// TwinCAT 3 PLC project Stream_lib
// Title: Stream_lib
// Company: Chua Siang Poh
// Author: Chua Siang Poh
// ProjectVersion: 1.1
// ProgramVersion: 3.1.4020.10
// libraries:
//   Tc2_Standard, * (Beckhoff Automation GmbH)
//   Tc2_System, * (Beckhoff Automation GmbH)
//   Tc3_Module, * (Beckhoff Automation GmbH)
// project tree:
//   Base Component/Class/Binary/ C_BINARYREADER.TcPOU, C_BINARYWRITER.TcPOU
//   Base Component/Class/HTTP/Datatype/ E_HTTP_CODEGROUP.TcDUT, E_HTTP_CONNECTION.TcDUT, E_HTTP_VERB.TcDUT, T_HTTP_BODY.TcDUT, T_HTTP_URL.TcDUT
//   Base Component/Class/HTTP/Functions/ GET_URL_LENGTH.TcPOU
//   Base Component/Class/HTTP/ GVL_HTTP_PARAMETERS.TcGVL
//   Base Component/Class/HTTP/Message/Base/ C_HTTP_MESSAGE.TcPOU
//   Base Component/Class/HTTP/Message/ C_HTTP_HEADER.TcPOU, C_HTTP_REQUEST.TcPOU, C_HTTP_RESPONSE.TcPOU
//   Base Component/Class/Stream/ C_BINARYSTREAM.TcPOU, C_FILESTREAM.TcPOU, C_HTTPSTREAM.TcPOU
//   Base Component/Datatype/ E_STREAMSEEKTYPE.TcDUT
//   Base Component/Interface/ I_STREAM.TcIO
//   Project Information/ F_GetCompany.TcPOU, F_GetTitle.TcPOU, F_GetVersion.TcPOU
//   Version/ Global_Version.TcGVL
// (motion and I/O tree: see PLC project motion_library)
// real-time tasks:
//   TASK PlcTask: cycle T#10ms, priority 20, ADS port 350

// ---- Base Component/Class/HTTP/Datatype/E_HTTP_CODEGROUP.TcDUT
{attribute 'qualified_only'}
{attribute 'strict'}
TYPE E_HTTP_CODEGROUP :
(
	E_GROUP_INFOMATION := 100,
	E_GROUP_SUCCESS := 200,
	E_GROUP_REDIRECTION := 300,
	E_GROUP_CLIENTERROR := 400,
	E_GROUP_SERVERERROR := 500
)UDINT;
END_TYPE

// ---- Base Component/Class/HTTP/Datatype/E_HTTP_CONNECTION.TcDUT
{attribute 'qualified_only'}
{attribute 'strict'}
TYPE E_HTTP_CONNECTION :
(
	E_CONNECTION_CLOSE := 0,
	E_CONNECTION_KEEP_ALIVE
);
END_TYPE

// ---- Base Component/Class/HTTP/Datatype/E_HTTP_VERB.TcDUT
{attribute 'qualified_only'}
{attribute 'strict'}
TYPE E_HTTP_VERB :
(
	E_HTTP_REQUEST_GET := 0,
	E_HTTP_REQUEST_POST,
	E_HTTP_REQUEST_DELETE,
	E_HTTP_REQUEST_PUT,
	E_HTTP_REQUEST_HEAD,
	E_HTTP_REQUEST_CONNECT,
	E_HTTP_REQUEST_OPTIONS,
	E_HTTP_REQUEST_TRACE
)UDINT;
END_TYPE

// ---- Base Component/Class/HTTP/Datatype/T_HTTP_BODY.TcDUT
TYPE T_HTTP_BODY : ARRAY[0..GVL_HTTP_PARAMETERS.MAX_HTTP_BODY_LENGTH] OF BYTE; END_TYPE

// ---- Base Component/Class/HTTP/Datatype/T_HTTP_URL.TcDUT
TYPE T_HTTP_URL : STRING(GVL_HTTP_PARAMETERS.MAX_HTTP_URL_LENGTH); END_TYPE

// ---- Base Component/Datatype/E_STREAMSEEKTYPE.TcDUT
{attribute 'qualified_only'}
{attribute 'strict'}
TYPE E_STREAMSEEKTYPE :
(
	Origin := 0,
	Current,
	End
);
END_TYPE

// ---- Base Component/Class/HTTP/GVL_HTTP_PARAMETERS.TcGVL
{attribute 'qualified_only'}
VAR_GLOBAL CONSTANT
	MAX_HTTP_BODY_LENGTH 	: UDINT := 30000;
	MAX_HTTP_URL_LENGTH 	: UDINT := 1000;
END_VAR

// ---- Version/Global_Version.TcGVL
{attribute 'TcGenerated'}
// This function has been automatically generated from the project information.
VAR_GLOBAL CONSTANT
	{attribute 'const_non_replaced'}
	{attribute 'linkalways'}
	stLibVersion_Stream_lib : ST_LibVersion := (iMajor := 1, iMinor := 1, iBuild := 0, iRevision := 0, sVersion := '1.1');
END_VAR

// ---- Base Component/Interface/I_STREAM.TcIO
INTERFACE I_STREAM

PROPERTY BufferSize : UDINT
GET
END_GET
END_PROPERTY

METHOD Close : DINT
VAR_INPUT
END_VAR
END_METHOD

PROPERTY EndOfStream : BOOL
GET
END_GET
END_PROPERTY

PROPERTY IsValid : BOOL
GET
END_GET
END_PROPERTY

METHOD Peek : DINT
VAR_INPUT
	ptr_DataOut : POINTER TO BYTE;
END_VAR
END_METHOD

PROPERTY Position : UDINT
GET
END_GET
END_PROPERTY

METHOD Read : DINT
VAR_INPUT
	ptr_DataOut : PVOID;
	Length		: UDINT;
END_VAR
END_METHOD

METHOD Seek : DINT
VAR_INPUT
	Offset 		: UDINT;
	SeekStyle 	: E_STREAMSEEKTYPE;
END_VAR
END_METHOD

METHOD Write : DINT
VAR_INPUT
	ptr_DataIn	: PVOID;
	Length		: UDINT;
END_VAR
END_METHOD

END_INTERFACE

// ---- Base Component/Class/Binary/C_BINARYREADER.TcPOU
FUNCTION_BLOCK C_BINARYREADER
VAR_INPUT
END_VAR
VAR_OUTPUT
END_VAR
VAR
	_BASESTREAM 	: I_STREAM;
END_VAR

PROPERTY BASE_STREAM : I_STREAM
GET
Base_Stream := _BASESTREAM;
END_GET
END_PROPERTY

METHOD CLOSE : DINT
VAR_INPUT
END_VAR
Close := _BASESTREAM.Close();
_BASESTREAM := 0;
RETURN;
END_METHOD

METHOD NEW : DINT
VAR_INPUT
	STREAM : I_STREAM;
END_VAR
IF STREAM = 0 THEN
	New := 1;
	RETURN;
ELSE
	IF STREAM.IsValid THEN
		_BASESTREAM := STREAM;
		_BASESTREAM.Seek( 0, E_STREAMSEEKTYPE.Origin);
		New := -1;
		RETURN;
	ELSE
		New := 1;
		RETURN;
	END_IF
END_IF
END_METHOD

METHOD READ_BOOL : DINT
VAR_INPUT
	out_data : POINTER TO BOOL;
END_VAR
IF _BASESTREAM = 0 THEN
	Read_Bool := 1;
	RETURN;
END_IF

Read_Bool := _BASESTREAM.Read(out_data , 1);
RETURN;
END_METHOD

METHOD READ_BYTES : DINT
VAR_INPUT
	out_data 	: POINTER TO BYTE;
	length		: UDINT;
END_VAR
IF _BASESTREAM = 0 THEN
	Read_Bytes := 1;
	RETURN;
END_IF

Read_Bytes := _BASESTREAM.Read(out_data, length);
RETURN;
END_METHOD

METHOD READ_DOUBLE : DINT
VAR_INPUT
	out_data : POINTER TO LREAL;
END_VAR
IF _BASESTREAM = 0 THEN
	Read_Double := 1;
	RETURN;
END_IF

Read_Double := _BASESTREAM.Read(out_data , 8);
RETURN;
END_METHOD

METHOD READ_FLOAT : DINT
VAR_INPUT
	out_data : POINTER TO REAL;
END_VAR
IF _BASESTREAM = 0 THEN
	Read_Float := 1;
	RETURN;
END_IF

Read_Float := _BASESTREAM.Read(out_data , 4);
RETURN;
END_METHOD

METHOD READ_INT16 : DINT
VAR_INPUT
	out_data : POINTER TO INT;
END_VAR
IF _BASESTREAM = 0 THEN
	Read_Int16 := 1;
	RETURN;
END_IF

Read_Int16 := _BASESTREAM.Read(out_data , 2);
RETURN;
END_METHOD

METHOD READ_INT32 : DINT
VAR_INPUT
	out_data : POINTER TO DINT;
END_VAR
IF _BASESTREAM = 0 THEN
	Read_Int32 := 1;
	RETURN;
END_IF

Read_Int32 := _BASESTREAM.Read(out_data , 4);
RETURN;
END_METHOD

METHOD READ_STRING : DINT
VAR_INPUT
	out_data 	: PVOID;
	length		: UDINT;
END_VAR
IF _BASESTREAM = 0 THEN
	Read_String := 1;
	RETURN;
END_IF

Read_String := _BASESTREAM.Read(out_data, length);
RETURN;
END_METHOD

METHOD READ_UINT16 : DINT
VAR_INPUT
	out_data : POINTER TO UINT;
END_VAR
IF _BASESTREAM = 0 THEN
	Read_UInt16 := 1;
	RETURN;
END_IF

Read_UInt16 := _BASESTREAM.Read(out_data , 4);
RETURN;
END_METHOD

METHOD READ_UINT32 : DINT
VAR_INPUT
	out_data : POINTER TO UDINT;
END_VAR
IF _BASESTREAM = 0 THEN
	Read_UInt32 := 1;
	RETURN;
END_IF

Read_UInt32 := _BASESTREAM.Read(out_data , 4);
RETURN;
END_METHOD

END_FUNCTION_BLOCK

// ---- Base Component/Class/Binary/C_BINARYWRITER.TcPOU
FUNCTION_BLOCK C_BINARYWRITER
VAR_INPUT
END_VAR
VAR_OUTPUT
END_VAR
VAR
	_BASESTREAM 	: I_STREAM;
END_VAR

PROPERTY BASE_STREAM : I_STREAM
GET
Base_Stream := _BASESTREAM;
END_GET
END_PROPERTY

METHOD CLOSE : DINT
VAR_INPUT
END_VAR
Close := _BASESTREAM.Close();
_BASESTREAM := 0;
RETURN;
END_METHOD

METHOD NEW : DINT
VAR_INPUT
	STREAM : I_STREAM;
END_VAR
IF STREAM = 0 THEN
	New := 1;
	RETURN;
ELSE
	IF STREAM.IsValid THEN
		_BASESTREAM := STREAM;
		_BASESTREAM.Seek( 0, E_STREAMSEEKTYPE.Origin);
		New := -1;
		RETURN;
	ELSE
		New := 1;
		RETURN;
	END_IF
END_IF
END_METHOD

METHOD WRITE_BOOL : DINT
VAR_INPUT
	in_data : BOOL;
END_VAR
IF _BASESTREAM = 0 THEN
	Write_Bool := 1;
	RETURN;
END_IF

Write_Bool := _BASESTREAM.Write(ADR(in_data), 1);
RETURN;
END_METHOD

METHOD WRITE_BYTES : DINT
VAR_INPUT
	in_data 	: POINTER TO BYTE;
	length		: UDINT;
END_VAR
IF _BASESTREAM = 0 THEN
	Write_Bytes := 1;
	RETURN;
END_IF

Write_Bytes := _BASESTREAM.Write(in_data, length);
RETURN;
END_METHOD

METHOD WRITE_DOUBLE : DINT
VAR_INPUT
	in_data : LREAL;
END_VAR
IF _BASESTREAM = 0 THEN
	Write_Double := 1;
	RETURN;
END_IF

Write_Double := _BASESTREAM.Write(ADR(in_data), 8);
RETURN;
END_METHOD

METHOD WRITE_FLOAT : DINT
VAR_INPUT
	in_data : REAL;
END_VAR
IF _BASESTREAM = 0 THEN
	Write_Float := 1;
	RETURN;
END_IF

Write_Float := _BASESTREAM.Write(ADR(in_data) , 4);
RETURN;
END_METHOD

METHOD WRITE_INT16 : DINT
VAR_INPUT
	in_data : INT;
END_VAR
IF _BASESTREAM = 0 THEN
	Write_Int16 := 1;
	RETURN;
END_IF

Write_Int16 := _BASESTREAM.Write(ADR(in_data) , 2);
RETURN;
END_METHOD

METHOD WRITE_INT32 : DINT
VAR_INPUT
	in_data : DINT;
END_VAR
IF _BASESTREAM = 0 THEN
	Write_Int32 := 1;
	RETURN;
END_IF

Write_Int32 := _BASESTREAM.Write(ADR(in_data) , 4);
RETURN;
END_METHOD

METHOD WRITE_STRING : DINT
VAR_INPUT
	in_data 	: PVOID;
	length		: UDINT;
END_VAR
IF _BASESTREAM = 0 THEN
	Write_String := 1;
	RETURN;
END_IF

Write_String := _BASESTREAM.Write(in_data, length);
RETURN;
END_METHOD

METHOD WRITE_UINT16 : DINT
VAR_INPUT
	in_data : UINT;
END_VAR
IF _BASESTREAM = 0 THEN
	Write_UInt16 := 1;
	RETURN;
END_IF

Write_UInt16 := _BASESTREAM.Write(ADR(in_data) , 4);
RETURN;
END_METHOD

METHOD WRITE_UINT32 : DINT
VAR_INPUT
	in_data : UDINT;
END_VAR
IF _BASESTREAM = 0 THEN
	Write_UInt32 := 1;
	RETURN;
END_IF

Write_UInt32 := _BASESTREAM.Write(ADR(in_data) , 4);
RETURN;
END_METHOD

END_FUNCTION_BLOCK

// ---- Base Component/Class/HTTP/Functions/GET_URL_LENGTH.TcPOU
FUNCTION GET_URL_LENGTH : UDINT
VAR_INPUT
	PTR_URL : POINTER TO BYTE;
END_VAR
VAR
	I : UDINT;
END_VAR

FOR I := 0 TO GVL_HTTP_PARAMETERS.MAX_HTTP_URL_LENGTH BY 1 DO
	IF PTR_URL[I] = 0 THEN
		GET_URL_LENGTH := I;
		RETURN;
	END_IF
END_FOR
GET_URL_LENGTH := 0;
RETURN;

END_FUNCTION

// ---- Base Component/Class/HTTP/Message/Base/C_HTTP_MESSAGE.TcPOU
FUNCTION_BLOCK C_HTTP_MESSAGE
VAR_INPUT
END_VAR
VAR_OUTPUT
END_VAR
VAR
	//General header
		_CONNECTION 		: E_HTTP_CONNECTION;
	(*
		_CACHE_CONTROL		: STRING(255);
		_DATE 				: STRING(255);
		_PRAGMA				: STRING(255);
		_TRAILER 			: STRING(255);
		_TRANSFER_ENCODING	: STRING(255);
		_UPGRADE 			: STRING(255);
		_VIA 				: STRING(255);
		_WARNING 			: STRING(255);
	*)
	//Entity header
		_CONTENT_LENGTH		: UDINT;
	(*
		_ALLOW				: STRING(255);
		_CONTENT_ENCODING 	: STRING(255);
		_CONTENT_LANGUAGE 	: STRING(255);
		_CONTENT_MD5		: STRING(255);
		_CONTENT_TYPE		: STRING(255);
		_EXPIRES			: STRING(255);
		_LAST_MODIFIED		: STRING(255);
	*)
END_VAR

PROPERTY CONTENT_LENGTH : UDINT
GET
CONTENT_LENGTH := _CONTENT_LENGTH;
END_GET
SET
_CONTENT_LENGTH := CONTENT_LENGTH;
END_SET
END_PROPERTY

METHOD GET_BYTE : DINT
VAR_INPUT
	STREAM : I_STREAM;
END_VAR
VAR 
	_TERMINATOR 	: STRING(2) := '$R$N';
	HTTP_MESSAGE	: STRING(255);

	LENGTH 			: DINT;
END_VAR
IF STREAM = 0 THEN
	GET_BYTE := 1;
	RETURN;
END_IF

HTTP_MESSAGE := 'Connection: ';
IF STREAM.WRITE(ADR(HTTP_MESSAGE), LEN(HTTP_MESSAGE)) > 0 THEN
	GET_BYTE := 11;
	RETURN;
END_IF

CASE _CONNECTION OF 
E_HTTP_CONNECTION.E_CONNECTION_CLOSE:
	HTTP_MESSAGE := 'close';
E_HTTP_CONNECTION.E_CONNECTION_KEEP_ALIVE:
	HTTP_MESSAGE := 'keep-alive';
END_CASE
IF STREAM.WRITE(ADR(HTTP_MESSAGE), LEN(HTTP_MESSAGE)) > 0 THEN
	GET_BYTE := 12;
	RETURN;
END_IF

IF STREAM.WRITE(ADR(_TERMINATOR), LEN(_TERMINATOR)) > 0 THEN
	GET_BYTE := 13;
	RETURN;
END_IF

HTTP_MESSAGE := 'Content-Length: ';
IF STREAM.WRITE(ADR(HTTP_MESSAGE), LEN(HTTP_MESSAGE)) > 0 THEN
	GET_BYTE := 21;
	RETURN;
END_IF
HTTP_MESSAGE := UDINT_TO_STRING(_CONTENT_LENGTH);
IF STREAM.WRITE(ADR(HTTP_MESSAGE), LEN(HTTP_MESSAGE)) > 0 THEN
	GET_BYTE := 22;
	RETURN;
END_IF
IF STREAM.WRITE(ADR(_TERMINATOR), LEN(_TERMINATOR)) > 0 THEN
	GET_BYTE := 23;
	RETURN;
END_IF

GET_BYTE := -1;
RETURN;
END_METHOD

PROPERTY HTTP_CONNECTION : E_HTTP_CONNECTION
GET
HTTP_CONNECTION := _CONNECTION;
END_GET
SET
_CONNECTION := HTTP_CONNECTION;
END_SET
END_PROPERTY

END_FUNCTION_BLOCK

// ---- Base Component/Class/HTTP/Message/C_HTTP_HEADER.TcPOU
FUNCTION_BLOCK C_HTTP_HEADER
VAR_INPUT
END_VAR
VAR_OUTPUT
END_VAR
VAR
	_FIELD 	: STRING(255);
	_NAME 	: STRING(255);
END_VAR

PROPERTY FIELD : STRING(255)
GET
FIELD := _FIELD;
END_GET
SET
_FIELD := FIELD;
END_SET
END_PROPERTY

METHOD GET_STRING : STRING(GVL_HTTP_PARAMETERS.MAX_HTTP_HEADER_LENGTH)
VAR_INPUT
	LENGTH : POINTER TO DINT;
END_VAR
VAR
	_OFFSET 		: DINT	:= 0;
	_BUFFER_STRING 	: ARRAY[0..GVL_HTTP_PARAMETERS.MAX_HTTP_HEADER_LENGTH] OF BYTE;
	_DELIMITER 		: STRING(2) := ': ';
	_TERMINATOR		: STRING(2) := '$R$N';
END_VAR
MEMCPY(ADR(_BUFFER_STRING[_OFFSET]), ADR(_NAME), LEN(NAME));
_OFFSET := _OFFSET + LEN(NAME);
MEMCPY(ADR(_BUFFER_STRING[_OFFSET]), ADR(_DELIMITER), LEN(_DELIMITER));
_OFFSET := _OFFSET + LEN(_DELIMITER);
MEMCPY(ADR(_BUFFER_STRING[_OFFSET]), ADR(_FIELD), LEN(_FIELD));
_OFFSET := _OFFSET + LEN(_FIELD);
MEMCPY(ADR(_BUFFER_STRING[_OFFSET]), ADR(_TERMINATOR), LEN(_TERMINATOR));
_OFFSET := _OFFSET + LEN(_TERMINATOR);
LENGTH^ := _OFFSET;
MEMCPY(ADR(GET_STRING), ADR(_BUFFER_STRING), 515);
RETURN;
END_METHOD

PROPERTY NAME : STRING(255)
GET
NAME := _NAME;
END_GET
SET
_NAME := NAME;
END_SET
END_PROPERTY

METHOD PARSE : DINT
VAR_INPUT
END_VAR
END_METHOD

END_FUNCTION_BLOCK

// ---- Base Component/Class/HTTP/Message/C_HTTP_REQUEST.TcPOU
FUNCTION_BLOCK C_HTTP_REQUEST EXTENDS C_HTTP_MESSAGE
VAR_INPUT
END_VAR
VAR_OUTPUT
END_VAR
VAR
	_REQUEST 		: E_HTTP_VERB;
	
	_URL 			: T_HTTP_URL;
	
	_VERSION_MAJOR 	: UDINT := 1;
	_VERSION_MINOR 	: UDINT := 1;
	
	_HOST 				: STRING(255);
(*                    	
    _ACCEPT_CHARSET 	: STRING(255);
    _ACCEPT_ENCODING	: STRING(255);
    _ACCEPT_LANGUAGE	: STRING(255);
    _AUTHORIZATION		: STRING(255);
    _EXPECT				: STRING(255);
    _FROM 				: STRING(255);
    _IF_MATCH 			: STRING(255);
    _IF_MODIFIED_SINCE 	: STRING(255);
    _IF_NONE_MATCH 		: STRING(255);
    _IF_RANGE 			: STRING(255);
    _IF_UNMODIFIED_SINCE: STRING(255);
    _MAX_FORWARDS 		: STRING(255);
    _PROXY_AUTHORIZATION: STRING(255);
    _RANGE 				: STRING(255);
    _REFERER 			: STRING(255);
    _TE 				: STRING(255);
    _USER_AGENT 		: STRING(255);
*)
	_BODY			: T_HTTP_BODY;
	_BODY_STREAM	: C_HTTPSTREAM;
	
	_PARSER 		: C_HTTPSTREAM;
	_PARSE_STATE	: UDINT;
END_VAR

METHOD FB_init : BOOL
VAR_INPUT
	bInitRetains : BOOL; // if TRUE, the retain variables are initialized (warm start / cold start)
	bInCopyCode : BOOL;  // if TRUE, the instance afterwards gets moved into the copy code (online change)
END_VAR
_BODY_STREAM.NEW(ADR(_BODY), SIZEOF(_BODY));
END_METHOD

METHOD GET_BODY : I_STREAM
VAR_INPUT
END_VAR
GET_BODY := _BODY_STREAM;
END_METHOD

METHOD GET_BYTE : DINT
VAR_INPUT
	STREAM : I_STREAM;
END_VAR
VAR 
	_TERMINATOR 	: STRING(2) := '$R$N';
	HTTP_MESSAGE	: STRING(255);

	LENGTH 			: DINT;
END_VAR
IF STREAM = 0 THEN
	GET_BYTE := 1;
	RETURN;
END_IF

THIS^._CONTENT_LENGTH := _BODY_STREAM.POSITION;

//INSERT VERB
	CASE THIS^._REQUEST OF 
	E_HTTP_VERB.E_HTTP_REQUEST_GET:
		HTTP_MESSAGE := 'GET';
	E_HTTP_VERB.E_HTTP_REQUEST_CONNECT:
		HTTP_MESSAGE := 'CONNECT';
	E_HTTP_VERB.E_HTTP_REQUEST_DELETE:
		HTTP_MESSAGE := 'DELETE';
	E_HTTP_VERB.E_HTTP_REQUEST_HEAD:
		HTTP_MESSAGE := 'HEAD';
	E_HTTP_VERB.E_HTTP_REQUEST_OPTIONS:
		HTTP_MESSAGE := 'OPTIONS';
	E_HTTP_VERB.E_HTTP_REQUEST_POST:
		HTTP_MESSAGE := 'POST';
	E_HTTP_VERB.E_HTTP_REQUEST_PUT:
		HTTP_MESSAGE := 'PUT';
	E_HTTP_VERB.E_HTTP_REQUEST_TRACE:
		HTTP_MESSAGE := 'TRACE';
	END_CASE
	IF STREAM.WRITE(ADR(HTTP_MESSAGE), LEN(HTTP_MESSAGE)) > 0 THEN
		GET_BYTE := 10;
		RETURN;
	END_IF
	
//INSERT SPACE 
	HTTP_MESSAGE := ' ';
	IF STREAM.WRITE(ADR(HTTP_MESSAGE), LEN(HTTP_MESSAGE)) > 0 THEN
		GET_BYTE := 11;
		RETURN;
	END_IF
	
//INSERT URL
	IF STREAM.WRITE(ADR(_URL), GET_URL_LENGTH(ADR(_URL))) > 0 THEN
		GET_BYTE := 12;
		RETURN;
	END_IF
	HTTP_MESSAGE := ' ';
	IF STREAM.WRITE(ADR(HTTP_MESSAGE), LEN(HTTP_MESSAGE)) > 0 THEN
		GET_BYTE := 12;
		RETURN;
	END_IF
	
//INSERT VERSION
	HTTP_MESSAGE := 'HTTP/';	
	IF STREAM.WRITE(ADR(HTTP_MESSAGE), LEN(HTTP_MESSAGE)) > 0 THEN
		GET_BYTE := 13;
		RETURN;
	END_IF
	HTTP_MESSAGE := UDINT_TO_STRING(_VERSION_MAJOR);
	IF STREAM.WRITE(ADR(HTTP_MESSAGE), LEN(HTTP_MESSAGE)) > 0 THEN
		GET_BYTE := 13;
		RETURN;
	END_IF
	HTTP_MESSAGE := '.';
	IF STREAM.WRITE(ADR(HTTP_MESSAGE), LEN(HTTP_MESSAGE)) > 0 THEN
		GET_BYTE := 13;
		RETURN;
	END_IF
	HTTP_MESSAGE := UDINT_TO_STRING(_VERSION_MINOR);
	IF STREAM.WRITE(ADR(HTTP_MESSAGE), LEN(HTTP_MESSAGE)) > 0 THEN
		GET_BYTE := 13;
		RETURN;
	END_IF

//INSERT TERMINATOR
	HTTP_MESSAGE := '$R$N';
	IF STREAM.WRITE(ADR(HTTP_MESSAGE), LEN(HTTP_MESSAGE)) > 0 THEN
		GET_BYTE := 14;
		RETURN;
	END_IF
	
//INSERT STANDARD HEADERS
	HTTP_MESSAGE := 'Host: ';
	IF STREAM.WRITE(ADR(HTTP_MESSAGE), LEN(HTTP_MESSAGE)) > 0 THEN
		GET_BYTE := 21;
		RETURN;
	END_IF
	IF STREAM.WRITE(ADR(_HOST), LEN(_HOST)) > 0 THEN
		GET_BYTE := 21;
		RETURN;
	END_IF
	IF STREAM.WRITE(ADR(_TERMINATOR), LEN(_TERMINATOR)) > 0 THEN
		GET_BYTE := 21;
		RETURN;
	END_IF	

//INSERT COMMON HEADERS	
	IF SUPER^.GET_BYTE(STREAM) > 0 THEN
		GET_BYTE := 22;
		RETURN;
	END_IF
	
	{warning 'Not all stander headers implemented.'}

//INSERT USER HEADERS
	{warning 'User header not implemented yet.'}

//INSERT EXTRA TERMINATOR
	HTTP_MESSAGE := '$R$N';
	IF STREAM.WRITE(ADR(HTTP_MESSAGE), LEN(HTTP_MESSAGE)) > 0 THEN
		GET_BYTE := 29;
		RETURN;
	END_IF
	
//INSERT BODY
	IF STREAM.WRITE(ADR(_BODY), _BODY_STREAM.POSITION) > 0 THEN
		GET_BYTE := 31;
		RETURN;
	END_IF
	
GET_BYTE := -1;
RETURN;
END_METHOD

PROPERTY HOST : STRING(255)
GET
HOST := _HOST;
END_GET
SET
_HOST := HOST;
END_SET
END_PROPERTY

METHOD PARSE : DINT
VAR_INPUT
	PTR_DATA : PVOID;
	DATA_SIZE: UDINT;
END_VAR
VAR	

	_SPACE		: BYTE := 32; // ' '
	_FRONTSLASH	: BYTE := 47; // '/'
	_PERIOD		: BYTE := 46; // '.'
	_HEADDELIMIT: BYTE := 58; // ':'
	_CRLF		: ARRAY [0..1] OF BYTE := [13, 10];
	_CRLFCRLF	: ARRAY [0..3] OF BYTE := [13, 10, 13, 10];
	_LOCATION 	: UDINT;
	
	_VERB 		: ARRAY[0..80] OF BYTE;
	_VERBSTRING : STRING(10);
	
	_VERSIONSTRING : STRING(10);
	
	_HEADERSTRING	: STRING(255);
	//_HEADERWRITER	: C_STREAMWRITER;
	_SEGMENTBREAK	: UDINT;
	
	_ENDOFBODY	: BYTE := 0;
	STREAM: INT;
END_VAR
IF PTR_DATA = 0 OR DATA_SIZE = 0 THEN
	PARSE := 1;
	RETURN;
END_IF

CASE _PARSE_STATE OF
0:
	//Initialise
		_PARSER.Close();
		IF _PARSER.NEW(PTR_DATA, DATA_SIZE) > 0 THEN
			PARSE := 1;
			RETURN;
		END_IF
	//Parse Verb
		IF _PARSER.FIND(ADR(_SPACE), 1, ADR(_LOCATION)) < 0 THEN
			_PARSER.READ(ADR(_VERB), _LOCATION);
			CASE _LOCATION OF 
			3:
				_VERBSTRING := 'GET';
				IF MEMCMP(ADR(_VERBSTRING), ADR(_VERB), _LOCATION) <> 0 THEN
					_VERBSTRING := 'PUT';
					IF MEMCMP(ADR(_VERBSTRING), ADR(_VERB), _LOCATION) <> 0 THEN
						PARSE := 13;
						RETURN;
					END_IF
					_REQUEST := E_HTTP_VERB.E_HTTP_REQUEST_PUT;
				END_IF
				_REQUEST := E_HTTP_VERB.E_HTTP_REQUEST_GET;
			4:
				_VERBSTRING := 'POST';
				IF MEMCMP(ADR(_VERBSTRING), ADR(_VERB), _LOCATION) <> 0 THEN
					_VERBSTRING := 'HEAD';
					IF MEMCMP(ADR(_VERBSTRING), ADR(_VERB), _LOCATION) <> 0 THEN
						PARSE := 14;
						RETURN;
					END_IF
					_REQUEST := E_HTTP_VERB.E_HTTP_REQUEST_HEAD;
				END_IF
				_REQUEST := E_HTTP_VERB.E_HTTP_REQUEST_POST;
			5:
				_VERBSTRING := 'TRACE';
				IF MEMCMP(ADR(_VERBSTRING), ADR(_VERB), _LOCATION) <> 0 THEN
					PARSE := 15;
					RETURN;
				END_IF
				_REQUEST := E_HTTP_VERB.E_HTTP_REQUEST_TRACE;
			6:
				_VERBSTRING := 'DELETE';
				IF MEMCMP(ADR(_VERBSTRING), ADR(_VERB), _LOCATION) <> 0 THEN
					PARSE := 16;
					RETURN;
				END_IF
				_REQUEST := E_HTTP_VERB.E_HTTP_REQUEST_DELETE;
			7:
				_VERBSTRING := 'OPTIONS';
				IF MEMCMP(ADR(_VERBSTRING), ADR(_VERB), _LOCATION) <> 0 THEN
					_VERBSTRING := 'CONNECT';
					IF MEMCMP(ADR(_VERBSTRING), ADR(_VERB), _LOCATION) <> 0 THEN
						PARSE := 17;
						RETURN;
					END_IF
					_REQUEST := E_HTTP_VERB.E_HTTP_REQUEST_CONNECT;
				END_IF
				_REQUEST := E_HTTP_VERB.E_HTTP_REQUEST_OPTIONS;
			ELSE
				_PARSE_STATE := 0;
				PARSE := 10;
				RETURN;
			END_CASE
			_PARSER.SEEK(1, E_STREAMSEEKTYPE.Current);
		ELSE
			_PARSE_STATE := 0;
			PARSE := 1;
			RETURN;
		END_IF
		
	//Parse URL
		IF _PARSER.FIND(ADR(_SPACE), 1, ADR(_LOCATION)) < 0 THEN
			MEMSET(ADR(_URL), 0, SIZEOF(_URL));
			IF _PARSER.READ(ADR(THIS^._URL), _LOCATION) > 0 THEN
				_PARSE_STATE := 0;
				Parse := 20;
				RETURN;
			END_IF
			IF _PARSER.SEEK(1, E_STREAMSEEKTYPE.Current) > 0 THEN
				_PARSE_STATE := 0;
				Parse := 21;
				RETURN;
			END_IF
		ELSE
			_PARSE_STATE := 0;
			PARSE := 2;
			RETURN;
		END_IF
		
	//Parse Version
		_VERSIONSTRING := 'HTTP/';
		IF _PARSER.FIND(ADR(_VERSIONSTRING), 5, ADR(_LOCATION)) > 0 THEN
			_PARSE_STATE := 0;
			PARSE := 30;
			RETURN;
		ELSE
			IF _PARSER.SEEK(_LOCATION + 5, E_STREAMSEEKTYPE.Current) > 0 THEN
				_PARSE_STATE := 0;
				PARSE := 31;
				RETURN;
			END_IF
		END_IF
		IF _PARSER.FIND(ADR(_PERIOD), 1, ADR(_LOCATION)) < 0 THEN
			MEMSET(ADR(_VERSIONSTRING), 0, SIZEOF(_VERSIONSTRING));
			IF _PARSER.READ(ADR(_VERSIONSTRING), _LOCATION) > 0 THEN
				_PARSE_STATE := 0;
				PARSE := 32;
				RETURN;
			END_IF
			THIS^._VERSION_MAJOR := STRING_TO_UDINT(_VERSIONSTRING);
			IF _PARSER.SEEK(1, E_STREAMSEEKTYPE.Current) > 0 THEN
				_PARSE_STATE := 0;
				PARSE := 33;
				RETURN;
			END_IF
		ELSE
			_PARSE_STATE := 0;
			PARSE := 34;
			RETURN;
		END_IF
		IF _PARSER.FIND(ADR(_CRLF), 2, ADR(_LOCATION)) < 0 THEN
			MEMSET(ADR(_VERSIONSTRING), 0, SIZEOF(_VERSIONSTRING));
			IF _PARSER.READ(ADR(_VERSIONSTRING), _LOCATION) > 0 THEN
				_PARSE_STATE := 0;
				PARSE := 35;
				RETURN;
			END_IF
			THIS^._VERSION_MINOR := STRING_TO_UDINT(_VERSIONSTRING);
			IF _PARSER.SEEK(2, E_STREAMSEEKTYPE.Current) > 0 THEN
				_PARSE_STATE := 0;
				PARSE := 36;
				RETURN;
			END_IF
		ELSE
			_PARSE_STATE := 0;
			PARSE := 37;
			RETURN;
		END_IF
		_PARSE_STATE := _PARSE_STATE + 1;
		PARSE := 0;
		RETURN;
	_SEGMENTBREAK := 0;
1:
	{warning 'Implementation is not complete'}
	//Parse Headers
		WHILE TRUE DO 
			IF _PARSER.FIND(ADR(_CRLF), 2, ADR(_LOCATION)) < 0 THEN	
				IF _LOCATION = 0 THEN // Implies double CRLF is reached, ie. end of header
					EXIT;
				END_IF
				MEMSET(ADR(_HEADERSTRING), 0, SIZEOF(_HEADERSTRING));
				IF _PARSER.READ(ADR(_HEADERSTRING), _LOCATION) > 0 THEN
					_PARSE_STATE := 0;
					PARSE := 52;
					RETURN;
				END_IF
				IF _PARSER.SEEK(2, E_STREAMSEEKTYPE.Current) > 0 THEN
					_PARSE_STATE := 0;
					PARSE := 53;
					RETURN;
				END_IF
			ELSE
				_PARSE_STATE := 0;
				PARSE := 5; 
				RETURN;
			END_IF
			_SEGMENTBREAK := _SEGMENTBREAK + 1;
			IF _SEGMENTBREAK > 250 THEN
				_SEGMENTBREAK := 0;
				PARSE := 0;
				RETURN;
			END_IF
		END_WHILE
			
		IF _PARSER.SEEK(2, E_STREAMSEEKTYPE.Current) > 0 THEN
			_PARSE_STATE := 0;
			PARSE := 51;
			RETURN;
		ELSE
			_PARSE_STATE := _PARSE_STATE + 1;
			RETURN;
		END_IF
2:
	//Parse Body
		MEMSET(ADR(THIS^._BODY), 0, SIZEOF(_BODY));
		IF _PARSER.FIND(ADR(_ENDOFBODY), 1, ADR(_LOCATION)) < 0 THEN
			IF _PARSER.READ(ADR(THIS^._BODY), _LOCATION) > 0 THEN
				_PARSE_STATE := 0;
				PARSE := 60;
				RETURN;
			ELSE 
				_PARSE_STATE := 0;
				PARSE := -1;
				RETURN;
			END_IF
		ELSE
			_PARSE_STATE := 0;
			PARSE := 6;
			RETURN;
		END_IF
END_CASE

//Basic return, BUSY
PARSE := 0;
RETURN;
END_METHOD

PROPERTY URL : T_HTTP_URL
GET
URL := _URL;
END_GET
SET
_URL := URL;
END_SET
END_PROPERTY

PROPERTY VERB : E_HTTP_VERB
GET
VERB := _REQUEST;
END_GET
SET
_REQUEST := VERB;
END_SET
END_PROPERTY

END_FUNCTION_BLOCK

// ---- Base Component/Class/Stream/C_HTTPSTREAM.TcPOU
FUNCTION_BLOCK C_HTTPSTREAM IMPLEMENTS I_STREAM
VAR_INPUT
END_VAR
VAR_OUTPUT
END_VAR
VAR
	_BASE_MEM : POINTER TO BYTE;
	_BASE_SIZE: UDINT;
	
	_STREAM_POSITION : UDINT := 0;
END_VAR

PROPERTY BufferSize : UDINT
GET
END_GET
END_PROPERTY

METHOD Close : DINT
VAR_INPUT
END_VAR
_BASE_MEM := 0;
_BASE_SIZE:= 0;
_STREAM_POSITION := 0;
Close := -1;
RETURN;
END_METHOD

PROPERTY EndOfStream : BOOL
GET
EndOfStream := _STREAM_POSITION >= _BASE_SIZE;
END_GET
END_PROPERTY

PROPERTY IsValid : BOOL
GET
IsValid := _BASE_MEM <> 0;
END_GET
END_PROPERTY

METHOD NEW : DINT
VAR_INPUT
	PTR_BASE	: PVOID;
	BASE_SIZE	: UDINT;
END_VAR
IF PTR_BASE = 0 OR BASE_SIZE = 0 OR IsValid THEN
	NEW := 1;
	RETURN;
ELSE
	_BASE_MEM := PTR_BASE;
	_BASE_SIZE:= BASE_SIZE;
	_STREAM_POSITION := 0;
	NEW := -1;
	RETURN;
END_IF
END_METHOD

METHOD Peek : DINT
VAR_INPUT
	ptr_DataOut : POINTER TO BYTE;
END_VAR
IF NOT IsValid THEN
	Peek := 1;
	RETURN;
END_IF

ptr_DataOut^ := _BASE_MEM[_STREAM_POSITION];
Peek := -1;
RETURN;
END_METHOD

PROPERTY Position : UDINT
GET
Position := _STREAM_POSITION;
END_GET
END_PROPERTY

METHOD Read : DINT
VAR_INPUT
	ptr_DataOut : PVOID;
	Length		: UDINT;
END_VAR
IF NOT IsValid THEN
	Read := 1;
	RETURN;
END_IF

IF _STREAM_POSITION + Length > _BASE_SIZE THEN
	Read := 2;
	RETURN;
END_IF
		
MEMCPY(ptr_DataOut, _BASE_MEM + _STREAM_POSITION, Length);
_STREAM_POSITION := _STREAM_POSITION + Length;
READ := -1;
RETURN;
END_METHOD

METHOD Seek : DINT
VAR_INPUT
	Offset 		: UDINT;
	SeekStyle 	: E_STREAMSEEKTYPE;
END_VAR
IF NOT IsValid THEN
	Seek := 1;
	RETURN;
END_IF

CASE SeekStyle OF
	E_STREAMSEEKTYPE.Current_Reversed:
		IF OFFSET > _STREAM_POSITION THEN
			Seek := 2;
			RETURN;
		ELSE
			_STREAM_POSITION := _STREAM_POSITION - OFFSET;
			Seek := -1;
			RETURN;
		END_IF
	E_STREAMSEEKTYPE.Current:
		IF _STREAM_POSITION + OFFSET >= _BASE_SIZE THEN
			Seek := 2;
			RETURN;
		ELSE
			_STREAM_POSITION := _STREAM_POSITION + OFFSET;
			Seek := -1;
			RETURN;
		END_IF
	E_STREAMSEEKTYPE.End:
		IF OFFSET >= _BASE_SIZE THEN
			Seek := 2;
			RETURN;
		ELSE
			_STREAM_POSITION := _BASE_SIZE - Offset - 1;
			Seek := -1;
			RETURN;
		END_IF
	E_STREAMSEEKTYPE.Origin:
		IF OFFSET >= _BASE_SIZE THEN
			Seek := 2;
			RETURN;
		ELSE
			_STREAM_POSITION := Offset;
			Seek := -1;
			RETURN;
		END_IF
END_CASE
END_METHOD

METHOD Write : DINT
VAR_INPUT
	ptr_DataIn	: PVOID;
	Length		: UDINT;
END_VAR
IF NOT IsValid THEN
	Write := 1;
	RETURN;
END_IF

IF _STREAM_POSITION + Length > _BASE_SIZE THEN
	Write := 2;
	RETURN;
END_IF
		
MEMCPY(_BASE_MEM + _STREAM_POSITION, ptr_DataIn, Length);
_STREAM_POSITION := _STREAM_POSITION + Length;
Write := -1;
RETURN;
END_METHOD

END_FUNCTION_BLOCK

// ---- Base Component/Class/HTTP/Message/C_HTTP_RESPONSE.TcPOU
FUNCTION_BLOCK C_HTTP_RESPONSE EXTENDS C_HTTP_MESSAGE
VAR_INPUT
END_VAR
VAR_OUTPUT
END_VAR
VAR
	_CODEGROUP 		: E_HTTP_CODEGROUP := E_HTTP_CODEGROUP.E_GROUP_SUCCESS;
	_CODE			: UDINT := 0;
	
	_CODEMESSAGE	: STRING(255);
	
	_VERSION_MAJOR 	: UDINT := 1;
	_VERSION_MINOR 	: UDINT := 1;
	
(*
	_ACCEPT_RANGES		: STRING(255);
	_AGE				: STRING(255);
	_E_TAG				: STRING(255);
	_LOCATION			: STRING(255);
	_PROXY_AUTHENTICATE	: STRING(255);
	_RETRY_AFTER		: STRING(255);
	_SERVER				: STRING(255);
	_SET_COOKIE			: STRING(255);
	_VARY				: STRING(255);
	_WWW_AUTHENTICATE	: STRING(255);
*)

	_BODY 			: T_HTTP_BODY;
	_BODY_STREAM	: C_HTTPSTREAM;
END_VAR

METHOD FB_init : BOOL
VAR_INPUT
	bInitRetains : BOOL; // if TRUE, the retain variables are initialized (warm start / cold start)
	bInCopyCode : BOOL;  // if TRUE, the instance afterwards gets moved into the copy code (online change)
END_VAR
_BODY_STREAM.NEW(ADR(_BODY), SIZEOF(_BODY));
END_METHOD

METHOD GET_BYTE : DINT
VAR_INPUT
	STREAM : I_STREAM;
END_VAR
VAR 
	_RETURNCODE 	: UDINT;	

	_TERMINATOR 	: STRING(2) := '$R$N';
	_SPACE			: STRING(1) := ' ';
	
	HTTP_MESSAGE	: STRING(255);

	LENGTH 			: DINT;
END_VAR
IF STREAM = 0 THEN
	GET_BYTE := 1;
	RETURN;
END_IF

THIS^._CONTENT_LENGTH := _BODY_STREAM.POSITION;

//INSERT VERSION
	HTTP_MESSAGE := 'HTTP/';
	IF STREAM.WRITE(ADR(HTTP_MESSAGE), LEN(HTTP_MESSAGE)) > 0 THEN
		GET_BYTE := 10;
		RETURN;
	END_IF
	HTTP_MESSAGE := UDINT_TO_STRING(_VERSION_MAJOR);
	IF STREAM.WRITE(ADR(HTTP_MESSAGE), LEN(HTTP_MESSAGE)) > 0 THEN
		GET_BYTE := 11;
		RETURN;
	END_IF
	HTTP_MESSAGE := '.';
	IF STREAM.WRITE(ADR(HTTP_MESSAGE), LEN(HTTP_MESSAGE)) > 0 THEN
		GET_BYTE := 12;
		RETURN;
	END_IF
	HTTP_MESSAGE := UDINT_TO_STRING(_VERSION_MINOR);
	IF STREAM.WRITE(ADR(HTTP_MESSAGE), LEN(HTTP_MESSAGE)) > 0 THEN
		GET_BYTE := 13;
		RETURN;
	END_IF
	
	IF STREAM.WRITE(ADR(_SPACE), LEN(_SPACE)) > 0 THEN
		GET_BYTE := 14;
		RETURN;
	END_IF	
//RESPONSE CODE
	_RETURNCODE := _CODEGROUP; 
	_RETURNCODE := _RETURNCODE + _CODE;
	HTTP_MESSAGE := UDINT_TO_STRING(_RETURNCODE);
	IF STREAM.WRITE(ADR(HTTP_MESSAGE), LEN(HTTP_MESSAGE)) > 0 THEN
		GET_BYTE := 21;
		RETURN;
	END_IF
	
	IF STREAM.WRITE(ADR(_SPACE), LEN(_SPACE)) > 0 THEN
		GET_BYTE := 20;
		RETURN;
	END_IF
	
//RESPONSE MESSAGE
	IF STREAM.WRITE(ADR(_CODEMESSAGE), LEN(_CODEMESSAGE)) > 0 THEN
		GET_BYTE := 22;
		RETURN;
	END_IF

//INSERT TERMINATOR
	HTTP_MESSAGE := '$R$N';
	IF STREAM.WRITE(ADR(HTTP_MESSAGE), LEN(HTTP_MESSAGE)) > 0 THEN
		GET_BYTE := 23;
		RETURN;
	END_IF
	
//INSERT STANDARD HEADERS
	
	IF SUPER^.GET_BYTE(STREAM) > 0 THEN
		GET_BYTE := 31;
		RETURN;
	END_IF
	
	{warning 'Not all stander headers implemented.'}

//INSERT USER HEADERS
	{warning 'User header not implemented yet.'}

//INSERT TERMINATOR
	HTTP_MESSAGE := '$R$N';
	IF STREAM.WRITE(ADR(HTTP_MESSAGE), LEN(HTTP_MESSAGE)) > 0 THEN
		GET_BYTE := 30;
		RETURN;
	END_IF
	
//INSERT BODY
	IF STREAM.WRITE(ADR(_BODY), _BODY_STREAM.POSITION) > 0 THEN
		GET_BYTE := 41;
		RETURN;
	END_IF
	
GET_BYTE := -1;
RETURN;
END_METHOD

METHOD GET_STREAM : I_STREAM
VAR_INPUT
END_VAR
GET_STREAM := _BODY_STREAM;
END_METHOD

PROPERTY RESPONSE_CODE : UDINT
GET
RESPONSE_CODE := _CODE;
END_GET
SET
_CODE := RESPONSE_CODE;
END_SET
END_PROPERTY

PROPERTY RESPONSE_MESSAGE : STRING(255)
GET
RESPONSE_MESSAGE := _CODEMESSAGE;
END_GET
SET
_CODEMESSAGE := RESPONSE_MESSAGE;
END_SET
END_PROPERTY

PROPERTY RESPONSE_TYPE : E_HTTP_CODEGROUP
GET
RESPONSE_TYPE := THIS^._CODEGROUP;
END_GET
SET
THIS^._CODEGROUP := RESPONSE_TYPE;
END_SET
END_PROPERTY

END_FUNCTION_BLOCK

// ---- Base Component/Class/Stream/C_BINARYSTREAM.TcPOU
FUNCTION_BLOCK C_BINARYSTREAM IMPLEMENTS I_STREAM
VAR_INPUT
END_VAR
VAR_OUTPUT
END_VAR
VAR
	_MEMBUFFER 	: POINTER TO BYTE;
	_POSITION				: UDINT;
	//_PERMISSIBLE_LIMIT 		: UDINT;
	_MEMSIZE	: UDINT;
END_VAR

PROPERTY BUFFER_SIZE : UDINT
GET
Buffer_Size := _MEMSIZE;
END_GET
END_PROPERTY

METHOD CLOSE : DINT
VAR_INPUT
END_VAR
IF _MEMBUFFER <> 0 THEN
	__DELETE(_MEMBUFFER);
	_MEMBUFFER := 0;
END_IF
_POSITION := 0;
_PERMISSIBLE_LIMIT := 0;
_MEMSIZE := 0;
END_METHOD

PROPERTY END_OF_STREAM : BOOL
GET
IF _MEMBUFFER <> 0 THEN
	End_Of_Stream := _POSITION >= _MEMSIZE;
ELSE
	End_Of_Stream := TRUE;
END_IF
END_GET
END_PROPERTY

METHOD FB_exit : BOOL
VAR_INPUT
	bInCopyCode : BOOL; // if TRUE, the exit method is called for exiting an instance that is copied afterwards (online change).
END_VAR
IF NOT bInCopyCode THEN
    CLOSE();
END_IF
END_METHOD

PROPERTY IS_VALID : BOOL
GET
Is_Valid := _MEMBUFFER <> 0;
END_GET
END_PROPERTY

METHOD NEW : DINT
VAR_INPUT
	StreamSize	: UDINT;
END_VAR
IF _MEMBUFFER <> 0 THEN
	__DELETE(_MEMBUFFER);
END_IF
_MEMSIZE 				:= StreamSize;
//_PERMISSIBLE_LIMIT	 	:= _MEMSIZE - 1;
_POSITION 				:= 0;
_MEMBUFFER 				:= __NEW(BYTE, _MEMSIZE);

New := -1;
RETURN;
END_METHOD

METHOD PEEK : DINT
VAR_INPUT
	ptr_DataOut	: POINTER TO BYTE;
END_VAR
IF EndOfStream THEN
	Peek := 1; 
	RETURN;
ELSE
	ptr_DataOut^ := _MEMBUFFER[_POSITION];
	Peek := -1;
	RETURN;
END_IF
END_METHOD

PROPERTY POSITION : UDINT
GET
POSITION := _POSITION;
END_GET
END_PROPERTY

METHOD READ : DINT
VAR_INPUT
	ptr_DataOut	: PVOID;
	Length		: UDINT;
END_VAR
IF End_Of_Stream THEN
	Read := 1;
	RETURN;
ELSE
	IF _POSITION + Length > _MEMSIZE THEN
		Read := 2;
		RETURN;
	ELSE
		MEMCPY(ptr_DataOut, _MEMBUFFER + _POSITION, Length);
		_POSITION := _POSITION + Length;
		Read := -1;
		RETURN;
	END_IF
END_IF
END_METHOD

METHOD SEEK : DINT
VAR_INPUT
	Offset		: UDINT;	//Permissible range is 0 upto the total buffer size - 1;
	SeekStyle	: E_STREAMSEEKTYPE;
END_VAR
CASE SeekStyle OF 
	//Offsets from the beginning of the stream
	E_STREAMSEEKTYPE.Origin:
		IF Offset > _MEMSIZE THEN
			Seek := 1;
			RETURN;
		ELSE
			_POSITION := Offset;
			Seek := -1;
			RETURN;
		END_IF
	//Offsets from the end of the stream
	E_STREAMSEEKTYPE.End:
		IF Offset > _MEMSIZE THEN
			Seek := 1;
			RETURN;
		ELSE
			_POSITION := (_MEMSIZE) - Offset;
			Seek := -1;
			RETURN;
		END_IF
	//Offsets from the current position of the stream
	E_STREAMSEEKTYPE.Current:
		IF _POSITION + Offset > _MEMSIZE THEN
			Seek := 1;
			RETURN;
		ELSE
			_POSITION := _POSITION + Offset;
			Seek := -1;
			RETURN;
		END_IF
END_CASE
END_METHOD

METHOD WRITE : DINT
VAR_INPUT
	ptr_DataIn	: PVOID;
	Length		: UDINT;
END_VAR
IF End_Of_Stream THEN
	Write := 1;
	RETURN;
ELSE
	IF _POSITION + Length > _MEMSIZE THEN
		Write := 2;
		RETURN;
	ELSE
		MEMCPY(_MEMBUFFER + _POSITION, ptr_DataIn, Length);
		_POSITION := _POSITION + Length;
		Write := -1;
		RETURN;
	END_IF
END_IF
END_METHOD

END_FUNCTION_BLOCK

// ---- Base Component/Class/Stream/C_FILESTREAM.TcPOU
FUNCTION_BLOCK C_FILESTREAM IMPLEMENTS I_STREAM
VAR_INPUT
END_VAR
VAR_OUTPUT
END_VAR
VAR
	_FBFILEEND 	: FB_EOF;
	
	_EOF		: BOOL;
END_VAR

PROPERTY BufferSize : UDINT
GET
END_GET
END_PROPERTY

{warning 'add method implementation'}
METHOD Close : DINT
END_METHOD

PROPERTY EndOfStream : BOOL
GET
EndOfStream := _EOF;
END_GET
END_PROPERTY

METHOD FB_exit : BOOL
VAR_INPUT
	bInCopyCode : BOOL; // if TRUE, the exit method is called for exiting an instance that is copied afterwards (online change).
END_VAR
IF NOT bInCopyCode THEN
    CLOSE();
END_IF
END_METHOD

PROPERTY IsValid : BOOL
GET
END_GET
END_PROPERTY

{warning 'add method implementation'}
METHOD Peek : DINT
VAR_INPUT
	ptr_DataOut	: POINTER TO BYTE;
END_VAR
END_METHOD

PROPERTY Position : UDINT
GET
END_GET
END_PROPERTY

METHOD Read : DINT
VAR_INPUT
	ptr_DataOut	: PVOID;
	Length	: UDINT;
END_VAR
_FBFILEEND(
	sNetId:= , 
	hFile:= , 
	bExecute:= , 
	tTimeout:= , 
	bBusy=> , 
	bError=> , 
	nErrId=> , 
	bEOF=> );
END_METHOD

{warning 'add method implementation'}
METHOD Seek : DINT
VAR_INPUT
	Offset	: UDINT;
	SeekStyle	: E_STREAMSEEKTYPE;
END_VAR
END_METHOD

{warning 'add method implementation'}
METHOD Write : DINT
VAR_INPUT
	ptr_DataIn	: PVOID;
	Length	: UDINT;
END_VAR
END_METHOD

END_FUNCTION_BLOCK

// ---- Project Information/F_GetCompany.TcPOU
// This function has been automatically generated from the project information.
{attribute 'signature_flag' := '1073741824'}
{attribute 'TcGenerated'}
FUNCTION F_GetCompany : WSTRING
VAR_INPUT
	
END_VAR

F_GetCompany := "Chua Siang Poh";

END_FUNCTION

// ---- Project Information/F_GetTitle.TcPOU
// This function has been automatically generated from the project information.
{attribute 'signature_flag' := '1073741824'}
{attribute 'TcGenerated'}
FUNCTION F_GetTitle : WSTRING
VAR_INPUT
	
END_VAR

F_GetTitle := "CustomVisu_Frames";

END_FUNCTION

// ---- Project Information/F_GetVersion.TcPOU
// This function has been automatically generated from the project information.
{attribute 'signature_flag' := '1073741824'}
{attribute 'TcGenerated'}
FUNCTION F_GetVersion : ST_LibVersion
VAR_INPUT
	
END_VAR

F_GetVersion.iMajor := 0;
F_GetVersion.iMinor := 1;
F_GetVersion.iBuild := 0;
F_GetVersion.iRevision := 0;

END_FUNCTION
